TYPE E_AlarmType :
(
    None,
    BatteryLow,
    BatteryFull,
    GridFailure,
    NoGeneration,
    Emergency
);
END_TYPE

(* stored: Version 1.1.0.1, ProductVersion 3.1.4024.16
   DUT E_AlarmType: Id {fb3b0969-3ea3-4960-b71b-735df50e419a} *)
